// TIA Portal V19 export
FUNCTION_BLOCK "TYPIC_C501_IF_TME"   // FB60, FBD
TITLE = TYPIC_C501_IF_TME: Temperatuurmeting
{ S7_Optimized_Access := 'TRUE' }
AUTHOR : OCOTECH
FAMILY : Typical
NAME : C501.712
// Logisch Object Besturing: C501.712
// 
// De interne functie temperatuurmeting verzorgt de interne besturing en bewaking van een temperatuurmeting.
// stored: MemoryReserve 10, SetENOAutomatically false
   VAR_INPUT
      EXT_HW { ExternalAccessible := 'False'; ExternalVisible := 'False'; ExternalWritable := 'False'} : Bool;   // Sturings hardware (PLC) bewaking (1 = OK)
      IN_MWA { ExternalAccessible := 'False'; ExternalVisible := 'False'; ExternalWritable := 'False'} : Word;   // Meetwaarde
      IN_AUT_C501 { ExternalAccessible := 'False'; ExternalVisible := 'False'; ExternalWritable := 'False'} : Bool;   // Beveiligingen: serie geschakelde terugmelding (1= OK)
      CFG_MAX_SWA { ExternalAccessible := 'False'; ExternalVisible := 'False'; ExternalWritable := 'False'} : Real;   // Maximale waarde temperatuurmeting
      CFG_MIN_SWA { ExternalAccessible := 'False'; ExternalVisible := 'False'; ExternalWritable := 'False'} : Real;   // Minimale waarde temperatuurmeting
   END_VAR
   VAR_OUTPUT
      VAR_IF_TME { ExternalAccessible := 'False'; ExternalVisible := 'False'; ExternalWritable := 'False'} : "C501_VAR_IF_TME_TYPIC";   // Struct met alle variabelen naar bovenliggende functies
   END_VAR
   VAR
      STO { ExternalWritable := 'False'} : Struct   // Storingen
         A001 : Bool;   // Beveiliging aangesproken
         A002 : Bool;   // Draadbreuk analoge meting
         A003 : Bool;   // Meetbereik overschreden
         A004 : Bool;   // Temperatuurmeter geeft storing
      END_STRUCT;
      VAR { ExternalWritable := 'False'} : Struct   // Variabelen
         MWA : Real;   // Meetwaarde
         EXT_HW { ExternalAccessible := 'False'; ExternalVisible := 'False'} : Bool;   // Sturings hardware (PLC) in storing
      END_STRUCT;
   END_VAR
BEGIN

REGION Network 1: START
END_REGION

REGION Network 2: +++ Verwerking analoge meting +++
   // Verwerking analoge meting naar een meetwaarde in m3/u en detectie storingen van de meting.
END_REGION

REGION Network 3: +++ Storingen +++
   // Storingen van de analoge meting.
END_REGION

REGION Network 4: Storing A001: Beveiliging aangesproken
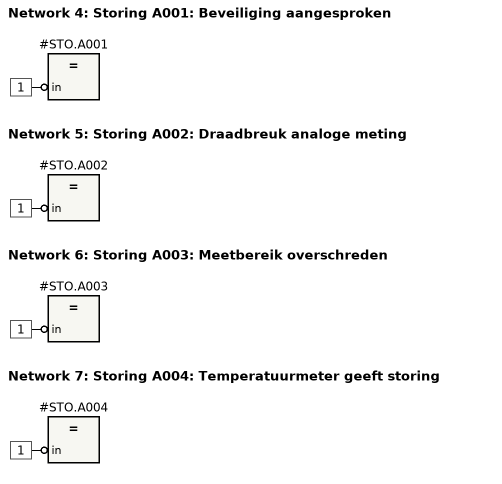
   #STO.A001 := NOT 1;
END_REGION

REGION Network 5: Storing A002: Draadbreuk analoge meting
   #STO.A002 := NOT 1;
END_REGION

REGION Network 6: Storing A003: Meetbereik overschreden
   #STO.A003 := NOT 1;
END_REGION

REGION Network 7: Storing A004: Temperatuurmeter geeft storing
   #STO.A004 := NOT 1;
END_REGION

REGION Network 8 (SCL): EINDE
   // Variabelen van intern scada rakvlak naar outputs copieren
   #VAR_IF_TME.MWA := #VAR.MWA;
   #VAR_IF_TME.EXT_HW := #VAR.EXT_HW;
   #VAR_IF_TME.STO := #STO;
END_REGION
END_FUNCTION_BLOCK
